# EPICS substitutions: examples/test/el6002/ecmcEL6002_custom.substitutions
file "ecmcEcSlave.template"
{
  pattern {}
          {}
}

file "ecmcEL6002-chX_custom.template"
{
  pattern {CH_ID, NELM }
          {01,    22   }
          {02,    22   }
}
